FUNCTION_BLOCK OneVSD_Latch
VAR_INPUT
	VSD_Run: BOOL;
	VSD_Fault: BOOL;
	VSD_Delay: TIME;
	OA_VSDReset: BOOL;
	
END_VAR
VAR_OUTPUT
	VSD_FaultAct: BOOL;
END_VAR
VAR
	T1:TON;
END_VAR

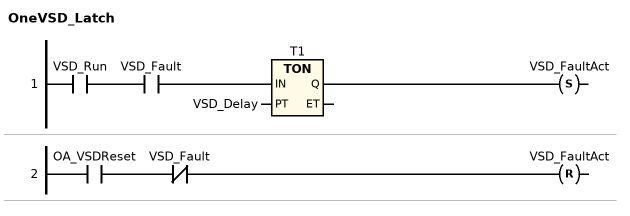
// NETWORK 1
T1(IN := VSD_Run AND VSD_Fault, PT := VSD_Delay); // TON
VSD_FaultAct S= T1.Q;

// NETWORK 2
VSD_FaultAct R= OA_VSDReset AND NOT VSD_Fault;

END_FUNCTION_BLOCK

(* stored: Version 1.1.0.1, ProductVersion 3.1.4024.12
   POU OneVSD_Latch: Id {5df5db4a-a480-4d7b-ab0e-b2aa3f1b8fea}, SpecialFunc None *)
